// TIA Portal V20 export
TYPE "LER_typeBrakeTestUnitMonitoring"
// stored: Access Published
   STRUCT
      emStatus { S7_SetPoint := 'True'} : "LER_typeBrakeTestEmStatus";
      error { ExternalWritable := 'False'} : Bool;
      allReady { ExternalWritable := 'False'} : Bool;
      allBusy { ExternalWritable := 'False'} : Bool;
      allComplete { ExternalWritable := 'False'} : Bool;
      firstScan { ExternalWritable := 'False'} : Bool;
      after8Hours { ExternalWritable := 'False'} : Bool;
      after24Hours { ExternalWritable := 'False'} : Bool;
   END_STRUCT;
END_TYPE
